FUNCTION IsNone : BOOL
VAR_INPUT
	eResult			: Result;
END_VAR
VAR_OUTPUT
	eCarry			: Result;
END_VAR

IsNone := eResult = 0;
eCarry := eResult;

END_FUNCTION

(* stored: Version 1.1.0.1
   POU IsNone: Id {45d926e7-4340-49c1-9630-09ea933bc1ee}, SpecialFunc None *)
